{attribute 'linkalways'} 
{attribute 'no_explicit_call' := 'This FB is a CLASS and must be accessed using methods or properties'}
{attribute 'enable_dynamic_creation'}
FUNCTION_BLOCK Node_F_VN_ConvertElementType EXTENDS VisionNode
VAR
    ipSrcImage : _ITcVnImage;
    ipDestImage : _ITcVnImage;
    eElementType : _ETcVnElementType(ETcVnElementType.TCVN_ET_SAME_AS_SOURCE);
    hrPrev : _HRESULT(S_OK);
	hresult : _HRESULT(S_OK);
END_VAR

METHOD PUBLIC  Clone : I_Node
VAR
	pNode : POINTER TO Node_F_VN_ConvertElementType;
END_VAR
pNode := __NEW(Node_F_VN_ConvertElementType);
Clone := pNode^;
END_METHOD

METHOD FB_init : BOOL
VAR_INPUT
	bInitRetains : BOOL; // if TRUE, the retain variables are initialized (warm start / cold start)
	bInCopyCode : BOOL;  // if TRUE, the instance afterwards gets moved into the copy code (online change)
END_VAR
AddInput('ipSrcImage', ipSrcImage);
AddInput('hrPrev', hrPrev);
AddParameter('eElementType', eElementType);
AddOutput('ipDestImage', ipDestImage);
AddOutput('hresult',hresult);
END_METHOD

METHOD PROTECTED OnExecute : HRESULT
hresult.Value := F_VN_ConvertElementType(
    ipSrcImage := ipSrcImage.Value,
	ipDestImage := ipDestImage.Value,
    eElementType := eElementType.Value,
	hrPrev:= hrPrev.Value);
END_METHOD

METHOD PUBLIC PreExecutionCheck
VAR_INPUT
	Check : I_PreExecutionChecks;
END_VAR
Check.IsTrue(ipSrcImage.IsValid, 'ipSrcImage must contain an image');
END_METHOD

END_FUNCTION_BLOCK

(* stored: Version 1.1.0.1, ProductVersion 3.1.4024.13
   POU Node_F_VN_ConvertElementType: Id {05ea1367-a053-005f-2303-49340c9a056c}, SpecialFunc None
   Folder Constructor: Id {9652d596-ff51-07c4-144f-2d01cf370a9a}
   Method Clone: Id {1a276de9-18c7-0912-172a-679197ffb1ac}
   Method FB_init: Id {1d6ced1b-c90d-077f-2aae-8b68ae2bb1d0}
   Method OnExecute: Id {592e5c49-75c3-023c-0ae1-833e2a887be1}
   Method PreExecutionCheck: Id {b13fecad-d80f-036d-0cfd-63b5f489c70b} *)
